FUNCTION_BLOCK LEDHMI (* Composite Function Block Type *)
  (* Standard: 61499-2 *)
  (* Version 0.0, 09/08/2022, Pranay Jhunjhunwala, UoA, template *)
  PACKAGE Main;
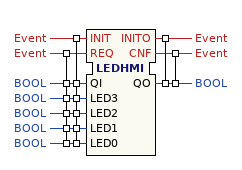
  EVENT_INPUT
    INIT WITH QI, LED3, LED2, LED1, LED0; (* Initialization Request *)
    REQ WITH QI, LED3, LED2, LED1, LED0; (* Normal Execution Request *)
  END_EVENT
  EVENT_OUTPUT
    INITO WITH QO; (* Initialization Confirm *)
    CNF WITH QO; (* Execution Confirmation *)
  END_EVENT
  VAR_INPUT
    QI : BOOL; (* Input event qualifier *)
    LED3 : BOOL;
    LED2 : BOOL;
    LED1 : BOOL;
    LED0 : BOOL;
  END_VAR
  VAR_OUTPUT
    QO : BOOL; (* Output event qualifier *)
  END_VAR
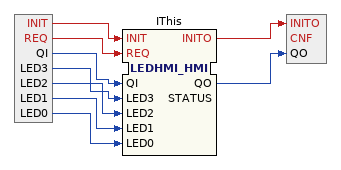
  FBS
    IThis : LEDHMI_HMI;
  END_FBS
  EVENT_CONNECTIONS
    INIT TO IThis.INIT;
    REQ TO IThis.REQ;
    IThis.INITO TO INITO;
  END_CONNECTIONS
  DATA_CONNECTIONS
    QI TO IThis.QI;
    LED3 TO IThis.LED3;
    LED2 TO IThis.LED2;
    LED1 TO IThis.LED1;
    LED0 TO IThis.LED0;
    IThis.QO TO QO;
  END_CONNECTIONS
END_FUNCTION_BLOCK
